// TIA Portal V19 export
DATA_BLOCK "TimeZones"   // DB13
{ S7_Optimized_Access := 'TRUE' }
// stored: MemoryReserve 100
   VAR
      UTC_0 : "Time Zone";
      UTC_1 { S7_SetPoint := 'True'} : "Time Zone";
      UTC_2 { S7_SetPoint := 'True'} : "Time Zone";
   END_VAR
BEGIN
   UTC_0.City := 'London';
   UTC_0.Offset := T#0H;
   UTC_1.City := 'Berlin';
   UTC_1.Offset := T#1H;
   UTC_2.City := 'Cairo';
   UTC_2.Offset := T#2H;
END_DATA_BLOCK
